(* PLC project Senza_nome, Sconosciuto Senza_nome 1 *)
(* stored: creationDateTime 2024-07-29T17:39:24, modificationDateTime 2024-07-30T08:59:42 *)

FUNCTION_BLOCK valves_handler
  VAR_INPUT
    IN1 : INT;
    STOP : BOOL;
    IN_TLB1 : INT;
    IN_TLB2 : INT;
  END_VAR
  VAR_OUTPUT
    OUT_MV1 : BOOL;
    OUT_MV2 : BOOL;
  END_VAR
  VAR
    real_value : INT;
  END_VAR

            
real_value :=  IN1 - 5;

if real_value <= IN_TLB2 then
  OUT_MV2 := FALSE;
  OUT_MV1 := TRUE;
end_if;

if real_value >= IN_TLB1 THEN
  OUT_MV2 := TRUE;
  OUT_MV1 := FALSE;
end_if;

if STOP = TRUE then
  OUT_MV2 := FALSE;
  OUT_MV1 := FALSE;
end_if;



          
END_FUNCTION_BLOCK

PROGRAM program0
  VAR_INPUT
    TLB2 : INT;
    TLB1 : INT;
    STOP : BOOL;
    START : BOOL;
    IN1 : INT;
    VALUE : INT;
  END_VAR
  VAR_OUTPUT
    MV1 : BOOL;
    MV2 : BOOL;
    CYCLE_ON : BOOL;
  END_VAR
  VAR
    valves_handler0 : valves_handler;
  END_VAR
  VAR  (* added by the conversion: wires and edge detectors of the diagram *)
    _EQ34_ENO : BOOL;
    _EQ34_OUT : BOOL;
  END_VAR

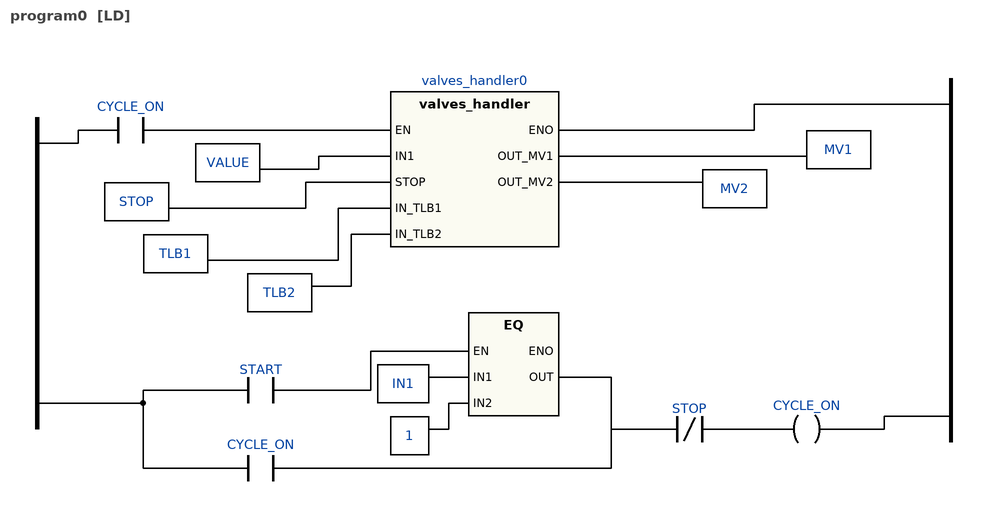
(* LD diagram, written out as Structured Text *)
valves_handler0(EN := CYCLE_ON, IN1 := VALUE, STOP := STOP, IN_TLB1 := TLB1, IN_TLB2 := TLB2);
IF valves_handler0.ENO THEN MV1 := valves_handler0.OUT_MV1; END_IF;
IF valves_handler0.ENO THEN MV2 := valves_handler0.OUT_MV2; END_IF;
_EQ34_OUT := EQ(EN := START, IN1 := IN1, IN2 := 1, ENO => _EQ34_ENO);
CYCLE_ON := (CYCLE_ON OR _EQ34_OUT) AND NOT STOP;
END_PROGRAM

CONFIGURATION Config0
  RESOURCE Res0 ON PLC
    TASK task0(INTERVAL := T#20ms, PRIORITY := 0);
    PROGRAM instance0 WITH task0 : program0;
  END_RESOURCE
END_CONFIGURATION
